RoboDK station: main.rdk

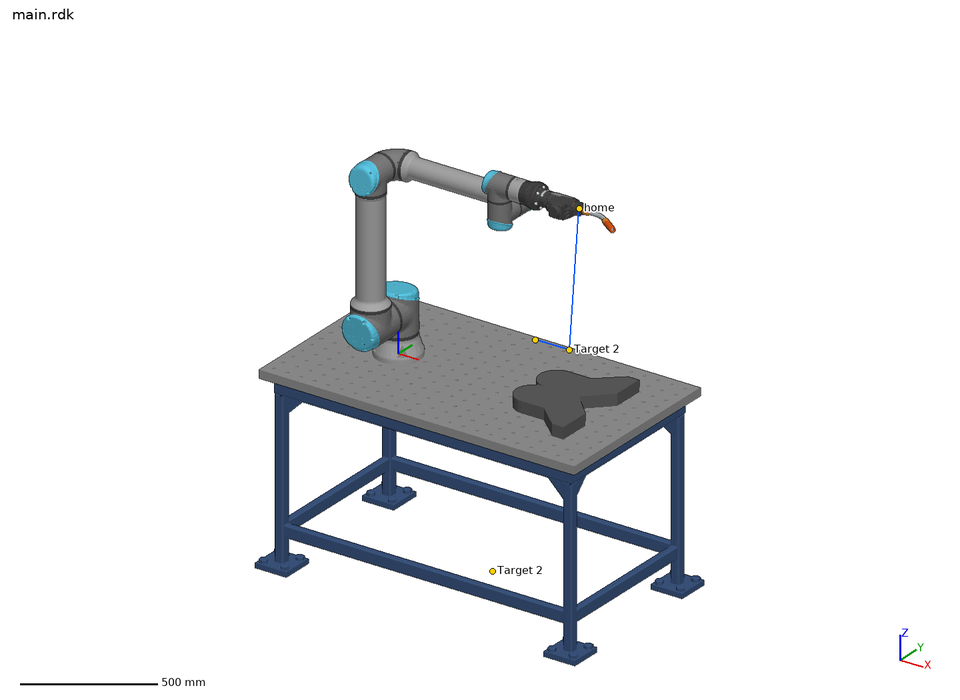
[picture v0: the station drawn from its stored meshes, robots at their saved joint values, targets as dots, program paths as lines]
Station main (saved by RoboDK 5.9.2). Poses are relative to the parent item; angles as X-Y-Z fixed-axis rotations.
  - frame UR10e Base at (0, 0, 0) mm
    - robot UR10e: 6 axes, payload 10 kg, reach 1300 mm, repeatability 0.05 mm, weight 28.9 kg
        modified DH rows (alpha deg, a mm, theta deg, d mm): 0, 0, 0, 180.7; 90, 0, 180, 0; 0, 612.6, 0, 0; 0, 571.335, 0, 174.15; -90, 0, 0, 119.85; 90, 0, 180, 116.55
        joint limits [-360, -360, -360, -360, -360, -360] to [360, 360, 360, 360, 360, 360]; home [0, -90, -90, 0, 90, 0]; saved at [0, -90, -90, 0, 90, 0]
      - tool Fronius MTB500i Welding Gun, TCP at (86, 0, 451.5) mm, rotated rx 97.62 ry 34.87 rz 12.87 deg, size 139 x 105 x 455.9 mm
    - target home (Cartesian target) at (924.38, -174.15, 913.15) mm, rotated rx -90 ry 0 rz -90 deg; joints [0, -90, -90, 0, 90, 0] of UR10e
    - target Target 2 (Cartesian target) at (810, -72, 270) mm, rotated rx 179.7 ry 40.67 rz -84.62 deg; joints [-8.516, -110.394, -89.258, -82.369, 129.148, -18.294] of UR10e
    - target Target 3 (Cartesian target) at (660, -74, 270) mm, rotated rx 179.7 ry 40.67 rz -84.62 deg; joints [-10.43, -97.866, -104.966, -80.697, 128.724, -20.695] of UR10e
      - target Target 2 (Cartesian target) at (810, -72, 270) mm, rotated rx 179.7 ry 40.67 rz -84.62 deg; joints [-8.516, -110.394, -89.258, -82.369, 129.148, -18.294] of UR10e
    - target Target 5 (Cartesian target) at (810, -72, 270) mm, rotated rx 179.7 ry 40.67 rz -84.62 deg; joints [-8.516, -110.394, -89.258, -82.369, 129.148, -18.294] of UR10e
    - target Target 6 (Cartesian target) at (660, -74, 270) mm, rotated rx 179.7 ry 40.67 rz -84.62 deg; joints [-10.43, -97.866, -104.966, -80.697, 128.724, -20.695] of UR10e
    - target Target 7 (Cartesian target) at (810, -72, 270) mm, rotated rx 179.7 ry 40.67 rz -84.62 deg; joints [-8.516, -110.394, -89.258, -82.369, 129.148, -18.294] of UR10e
  - object Table 1400x800x800mm at (0, 0, 0) mm, size 1420 x 820 x 800 mm, geometry from Table.sld
  - object Random obj at (650, 0, 0) mm, size 325 x 240 x 50 mm, geometry from Random obj.step
  - object Random obj at (650, 0, 50) mm, rotated rx -180 ry 0 rz 0 deg, size 325 x 240 x 50 mm, geometry from Random obj.step
  - program Prog1 (11 instructions, listed below)
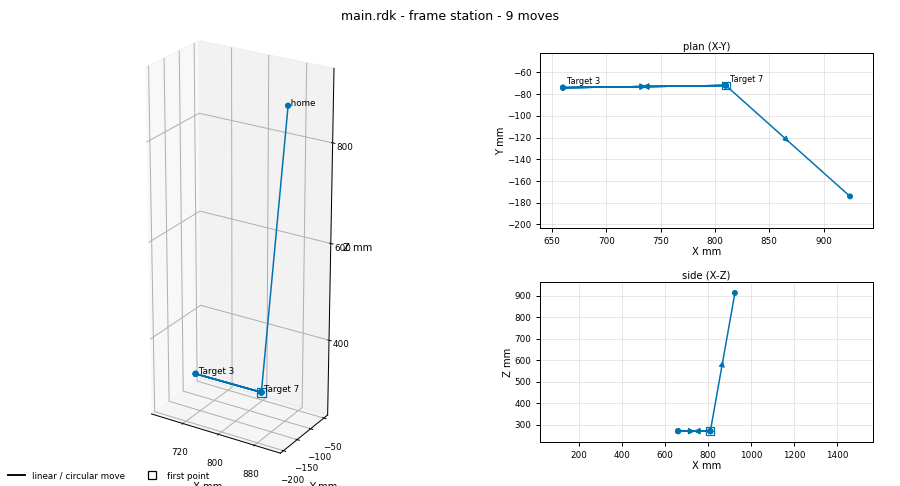
[picture p0: tool path of main.rdk in frame station, 9 of 9 moves have a stored position in this frame; points joined in program order, loops and branches not executed]

--- program Prog1 (robot UR10e) ---
  Set Ref.: UR10e Base
  Set Tool: ATI 9150-CDB-8-11-000 Deburring Tool (Spring) at (0, 0, 236.5) mm
  MoveJ (Target 7)
  MoveL (Target 2)
  MoveL (Target 3)
  MoveL (Target 5)
  MoveL (Target 6)
  MoveL (Target 7)
  MoveL (Target 3)
  MoveL (Target 5)
  MoveL (home)
